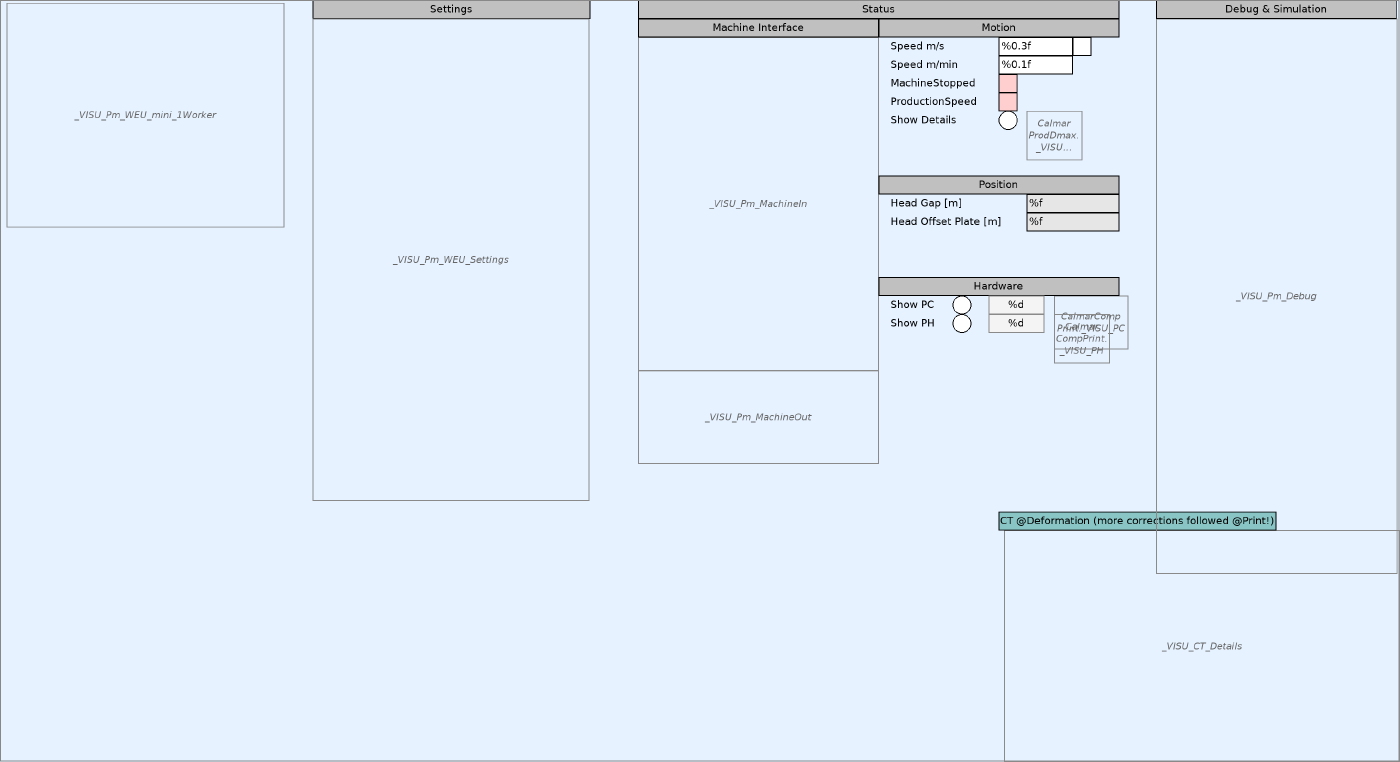
VISUALIZATION _VISU_Pm_WEU_1Worker  // 1514x825
VAR_IN_OUT
  mInst : FB_PrintModule_WEU;
END_VAR
    Frame (1086,574 428x251)
        shows _VISU_CT_Details(mInst := mInst.fbWorkerPrint[1])
    Rectangle (1080,554 300x20), "CT @Deformation (more corrections followed @Print!)"
    Frame (1140,320 80x58), invisible if: NOT mInst.fbView.bShowPcDetail
        shows CalmarCompPrint._VISU_PC(mInst := mInst._pPc[mInst.fbView.nSelPcDetail]^)
    Rectangle (960,340 110x20), "Show PH"
    Rectangle (960,320 110x20), "Show PC"
    Rectangle (960,40 120x20), "Speed m/s"
    Rectangle (1080,40 80x20), "%0.3f", text variable: mInst.fSpeed
    RoundedRectangle (1080,80 20x20), colour toggle: mInst.bMoving
    Rectangle (960,80 110x20), "MachineStopped"
    RoundedRectangle (1080,100 20x20), colour toggle: mInst.bSpeedReachedForPrinting
    Rectangle (960,100 110x20), "ProductionSpeed"
    Rectangle (960,60 120x20), "Speed m/min"
    Rectangle (1080,60 80x20), "%0.1f", text variable: mInst.fSpeedMpMin
    RoundedRectangle (1160,40 20x20), tooltip "Exeeds max. speed=%f", colour toggle: mInst._pModuleMachineFeedback^.bSpeedExeeded
        p4168582468: mInst._pModuleMachineFeedback^.fMaxSpeed
    Frame (690,401 260x101)
        shows _VISU_Pm_MachineOut(ref := mInst._pModuleMachineFeedback^)
    Frame (690,40 260x361)
        shows _VISU_Pm_MachineIn(ref := mInst._pModuleMachineState^)
    Rectangle (690,20 260x20), "Machine Interface"
    Rectangle (950,20 260x20), "Motion"
    Frame (7,3 300x243)
        shows _VISU_Pm_WEU_mini_1Worker(mInst := mInst)
    Rectangle (960,120 110x20), "Show Details"
    Ellipse (1080,120 20x20)
        toggle mInst.fbView.bShowPositionDetail
    Ellipse (1030,340 20x20)
        toggle mInst.fbView.bShowPhDetail
    Rectangle (950,300 260x20), "Hardware"
    Ellipse (1030,320 20x20)
        toggle mInst.fbView.bShowPcDetail
    Frame (1250,20 261x601), invisible if: NOT mInst.fbView.bShowDebugAndSim
        shows _VISU_Pm_Debug(mInst := mInst)
    Rectangle (338,0 300x20), "Settings"
    Rectangle (690,0 520x20), "Status"
    Rectangle (1250,0 260x20), "Debug & Simulation"
        toggle mInst.fbView.bShowDebugAndSim
    Rectangle (950,190 260x20), "Position"
    Rectangle (960,230 140x20), "Head Offset Plate [m]"
    Rectangle (1110,230 100x20), "%f", text variable: mInst.fC_HeadOffsetPlate
    Frame (1110,120 60x53), invisible if: NOT mInst.fbView.bShowPositionDetail
        shows CalmarProdDmax._VISU_PrintPositionDmax(m_Inst := mInst.fbPrintPosition)
    Frame (1140,340 60x53), invisible if: NOT mInst.fbView.bShowPhDetail
        shows CalmarCompPrint._VISU_PH(mInst := mInst._pPh[mInst.fbView.nSelPhDetail]^)
    Scrollbar (1069,340 60x20), "%d", text variable: mInst.fbView.nSelPhDetail, invisible if: NOT mInst.fbView.bShowPhDetail
        p2245068023: mInst._nPh
        p1057716461: mInst.fbView.nSelPhDetail
    Scrollbar (1069,320 60x20), "%d", text variable: mInst.fbView.nSelPcDetail, invisible if: NOT mInst.fbView.bShowPcDetail
        p2245068023: mInst._nPc
        p1057716461: mInst.fbView.nSelPcDetail
    Rectangle (1110,210 100x20), "%f", text variable: mInst._pModuleMachineFeedback^.fHeadGap
    Rectangle (960,210 140x20), "Head Gap [m]"
    Frame (338,20 299x522)
        shows _VISU_Pm_WEU_Settings(mInst := mInst)
END_VISUALIZATION

(* stored: Version 1.1.0.1, ProductVersion 3.1.4024.11
   Visu _VISU_Pm_WEU_1Worker: Id {509a8514-5119-4cda-ac8e-635dda5b6d1c} *)
